PROGRAM _FilterClean
VAR_INPUT
	i_bEnable				:BOOL;
	i_iFilterOn				:DINT;
	i_iFilterOff			:DINT;
END_VAR
VAR_OUTPUT
	q_bCmd					:BOOL;
END_VAR
VAR
	TON						:TON;
	TOF						:TOF;
END_VAR
VAR // added by the converter: edge detectors and wires of the graphical bodies
    _w1 : BOOL;
END_VAR

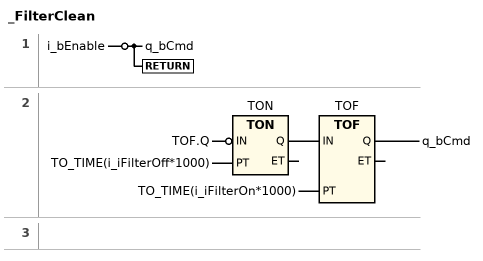
// NETWORK 1
_w1 := NOT i_bEnable;
q_bCmd := _w1;
IF _w1 THEN RETURN; END_IF

// NETWORK 2
TON(IN := NOT TOF.Q, PT := TO_TIME(i_iFilterOff*1000));
TOF(IN := TON.Q, PT := TO_TIME(i_iFilterOn*1000));
q_bCmd := TOF.Q;

// NETWORK 3

END_PROGRAM

(* stored: Version 1.1.0.1, ProductVersion 3.1.4024.12
   POU _FilterClean: Id {7ad454c7-e566-4446-ab2c-3a46974ef81f}, SpecialFunc None *)
